# EPICS substitutions: ek9000App/Db/EL5001.substitutions
file EL5001.template
{       pattern
        {
                TERMINAL,

        }
        {
        }
}
